// TIA Portal V16 export
// export: Created 2022-06-11T10:19:44.1245481Z, ExportSetting WithDefaults, DisplayName Totally Integrated Automation Portal, DisplayVersion V16 Update 3, DisplayName TIA Portal Version Control Interface, DisplayVersion V16 Update 2, DisplayName TIA Portal Openness, DisplayVersion V16 Update 3, DisplayName STEP 7 Professional, DisplayVersion V16 Update 3, DisplayName STEP 7 Safety, DisplayVersion V16, DisplayName WinCC Professional, DisplayVersion V16 Update 3
TYPE "UT31011_Dy_DevValve3Way"
TITLE = Dynamic UDT [DEVICE DRIVER] — Three-way Valve
// PRACTICAL SERIES AUTOMATION LIBRARY (PAL)   —   COPYRIGHT 2020 – M. GLEDHILL (MIT LICENCE)
//                   ———— ◆ ————
// FULL ONLINE DOCUMENTATION IS AVAILABLE AT: https://practicalseries.com/2001-pal/index.html
// stored: IsFailsafeCompliant false
   STRUCT
      revInfo : "UT01000_St_SysRevision";   // Revision information
      ___________0010_0 { ExternalAccessible := 'False'; ExternalVisible := 'False'; ExternalWritable := 'False'} : Int;
      ___________0010_1 { ExternalAccessible := 'False'; ExternalVisible := 'False'; ExternalWritable := 'False'} : Int;   // ▀▀▀▀ STATUS (FOR BLOCK ICON AND SYMBOL)
      status_Deenergised : Bool;   // STATUS — Valve is confirmed deenergised (1 = valve is in deenergised state)
      status_Energised : Bool;   // STATUS — Valve is confirmed energised (1 = valve is in energised state)
      status_Deenergising : Bool;   // STATUS — Valve is deenergising (1 = valve is deenergising, 0 = valve is not deenergising)
      status_Energising : Bool;   // STATUS — Valve is energising (1 = valve is energising, 0 = valve is not energising)
      status_Operating : Bool;   // STATUS — Valve is changing state (1 = valve is energising or deenergising, 0 = valve is not moving)
      status_Fault { ExternalWritable := 'False'} : Bool;   // STATUS — Valve is in fault (1 = fault present, 0 = healthy)
      status_OperateOn : Bool;   // STATUS — Valve output is on (1 = valve energised, 0 = valve deenergised)
      status_Aut : Bool;   // STATUS — Automatic mode active (1 = in automatic mode, 0 = not in automatic mode)
      status_Man : Bool;   // STATUS — Manual mode active (1 = in manual mode, 0 = not in manual mode)
      status_EStop : Bool;   // STATUS — E_STOP safety signal is active (1 = E_STOP active, 0 = E_STOP not active)
      status_Trip : Bool;   // STATUS — TRIP signal is active (1 = TRIP active, 0 = TRIP not active)
      status_Ilock : Bool;   // STATUS — INTERLOCK signal is active (1 = INTERLOCK active, 0 = INTERLOCK not active)
      status_Perm : Bool;   // STATUS — PERMISSIVE signal is active (1 = PERMISSIVE active, 0 = PERMISSIVE not active)
      status_BypassOn : Bool;   // STATUS — Valve is in bypass mode (1 = bypass mode on, 0 = normal)
      status_SimOn : Bool;   // STATUS — Valve is in simulation mode (1 = simulation mode on, 0 = normal)
      status_RemoteOn : Bool;   // STATUS — Valve is in remote mode (1 = remote mode, 0 = remote mode off)
      status_LocalOn : Bool;   // STATUS — Valve is in local mode (1 = local mode, 0 = local mode off)
      status_RLOff : Bool;   // STATUS — Remote/local mode disabled (1 = ALL mode on, 0 = RL mode selected)
      ___________0020_0 { ExternalAccessible := 'False'; ExternalVisible := 'False'; ExternalWritable := 'False'} : Int;
      ___________0020_1 { ExternalAccessible := 'False'; ExternalVisible := 'False'; ExternalWritable := 'False'} : Int;   // ▀▀▀▀ MESSAGES (ALARMS, WARNINGS, FAULTS AND EVENTS)
      msg_FailToEnergise : Bool;   // MESSAGE — Alarm – “Fail to energise” is active (1 = alarm active, 0 = alarm not active)
      msg_FailToDeenergise : Bool;   // MESSAGE — Alarm – “Fail to deenergise” is active (1 = alarm active, 0 = alarm not active)
      msg_FailWhileEnergised : Bool;   // MESSAGE — Alarm – “Fail while energised” is active (1 = alarm active, 0 = alarm not active)
      msg_FailWhileDeenergised : Bool;   // MESSAGE — Alarm – “Fail while deenergised” is active (1 = alarm active, 0 = alarm not active)
      msg_Flt_External : Bool;   // MESSAGE — Alarm – “External fault” is active (1 = alarm active, 0 = alarm not active)
      ___________0030_0 { ExternalAccessible := 'False'; ExternalVisible := 'False'; ExternalWritable := 'False'} : Int;
      ___________0030_1 { ExternalAccessible := 'False'; ExternalVisible := 'False'; ExternalWritable := 'False'} : Int;   // ▀▀▀▀ OPERATING MODE SELECTION (FROM FACEPLATE OR PANEL)
      mode_AutMan : Bool := true;   // MODE — Automatic or manual mode selection (1 = automatic mode, 0 = manual mode)
      mode_BypassOn : Bool;   // MODE — Bypass mode (1 = bypass mode active, 0 = normal)
      mode_SimOn : Bool;   // MODE — Simulation mode (1 = simulation mode active, 0 = normal)
      mode_SimValue : Int;   // MODE — Simulation value (0 no limits, 1 always open, 2 always closed, 3 follow demand)
      mode_RemoteOn : Bool;   // MODE — Local HMI control enabled (1 = control active, 0 = control disabled or N/A)
      mode_LocalOn : Bool;   // MODE — Remote SCADA control enabled (1 = control active, 0 = control disabled or N/A)
      mode_Reset : Bool;   // MODE — Fault reset (1 = Reset any faults – 1 cycle only, 0 = does nothing)
      ___________0040_0 { ExternalAccessible := 'False'; ExternalVisible := 'False'; ExternalWritable := 'False'} : Int;
      ___________0040_1 { ExternalAccessible := 'False'; ExternalVisible := 'False'; ExternalWritable := 'False'} : Int;   // ▀▀▀▀ CONTROL SIGNALS (TO OPERATE THE DEVICE)
      ctrl_Aut_EngDeng : Bool;   // CONTROL — Auto mode energise or deenergise valve (1 = energise in auto, 0 = deenergise in auto)
      ctrl_Man_EngDeng : Bool;   // CONTROL — Manual mode energise or deenergise valve (1 = energise in man, 0 = deenergise in man)
      ___________0050_0 { ExternalAccessible := 'False'; ExternalVisible := 'False'; ExternalWritable := 'False'} : Int;
      ___________0050_1 { ExternalAccessible := 'False'; ExternalVisible := 'False'; ExternalWritable := 'False'} : Int;   // ▀▀▀▀ BATCH AND BOOKING DATA
      batch_ID : UInt;   // BATCH — Booking ID (optional for batch operations)
      ___________0060_0 { ExternalAccessible := 'False'; ExternalVisible := 'False'; ExternalWritable := 'False'} : Int;
      ___________0060_1 { ExternalAccessible := 'False'; ExternalVisible := 'False'; ExternalWritable := 'False'} : Int;   // ▀▀▀▀ LIVE DATA (SCALED READING & TIMER VALUES)
      actual_Operating_Timer : Real;   // ACTUAL — Timer value — operating energising/deenergising timer actual value [seconds]
      actual_Last_Op_Time : Real;   // ACTUAL — Timer value — last operation time before feedback [seconds]
      ___________0090_0 { ExternalAccessible := 'False'; ExternalVisible := 'False'; ExternalWritable := 'False'} : Int;
      ___________0090_1 { ExternalAccessible := 'False'; ExternalVisible := 'False'; ExternalWritable := 'False'} : Int;   // ▀▀▀▀ BLOCK INTERNAL WORKING AND STORAGE AREA
      "$derived_fbk_eng" : Bool;   // INTERNAL — Derived feedback ENG signal (if CONFIG_FBK_ENG_EN = 0)
      "$derived_fbk_deng" : Bool;   // INTERNAL — Derived feedback DENG signal (if CONFIG_FBK_DENG_EN = 0)
      "$sim_fbk_eng" : Bool;   // INTERNAL — Simulated feedback ENG signal (if mode_SimOn = 1)
      "$sim_fbk_deng" : Bool;   // INTERNAL — Simulated feedback DENG signal (if mode_SimOn = 1)
      "$ctrl_EngDeng" : Bool;   // INTERNAL — actual energise or deenergise control signal passed to the valve (1 = eng, 0 = deng)
      "$pret_eng" : Bool;   // INTERNAL — Edge retention (+ve) rising edge of ctrl_OpenClose (change of state to energising)
      "$nret_deng" : Bool;   // INTERNAL — Edge retention (-ve) falling edge of ctrl_OpenClose (change of state to deenergising)
   END_STRUCT;
   // revInfo.REV_BLOCK := 'UT31011';
   // revInfo.REV_NUMBER := '000.801';
   // revInfo.REV_DATE := '2022.06.07';
   // revInfo.REV_AUTHOR := 'M. Gledhill';
END_TYPE
